// TIA Portal V19 export
FUNCTION "Analog_IN" : Void   // FC3, LAD
{ S7_Optimized_Access := 'TRUE' }
// stored: SetENOAutomatically false
BEGIN

REGION Network 1
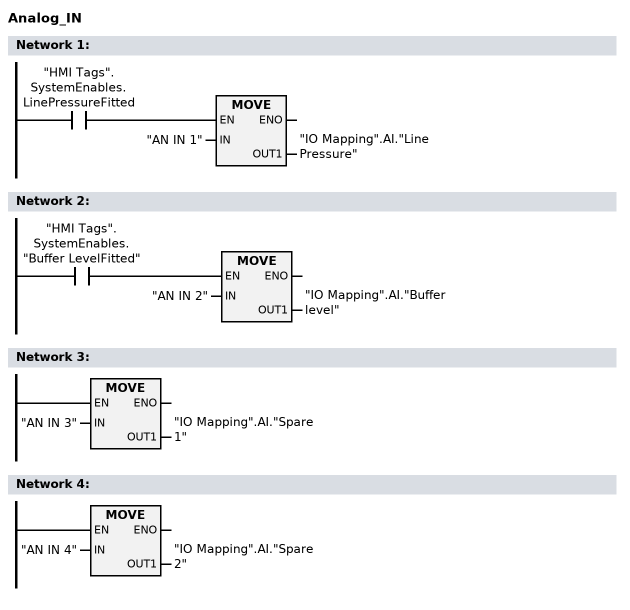
   RUNG wire#powerrail
      Contact( "HMI Tags".SystemEnables.LinePressureFitted )
      Move(in := "AN IN 1", out1 => "IO Mapping".AI."Line Pressure")
   END_RUNG
   // the same network as SCL:
   IF "HMI Tags".SystemEnables.LinePressureFitted THEN "IO Mapping".AI."Line Pressure" := "AN IN 1"; END_IF;
END_REGION

REGION Network 2
   RUNG wire#powerrail
      Contact( "HMI Tags".SystemEnables."Buffer LevelFitted" )
      Move(in := "AN IN 2", out1 => "IO Mapping".AI."Buffer level")
   END_RUNG
   // the same network as SCL:
   IF "HMI Tags".SystemEnables."Buffer LevelFitted" THEN "IO Mapping".AI."Buffer level" := "AN IN 2"; END_IF;
END_REGION

REGION Network 3
   RUNG wire#powerrail
      Move(in := "AN IN 3", out1 => "IO Mapping".AI."Spare 1")
   END_RUNG
   // the same network as SCL:
   "IO Mapping".AI."Spare 1" := "AN IN 3";
END_REGION

REGION Network 4
   RUNG wire#powerrail
      Move(in := "AN IN 4", out1 => "IO Mapping".AI."Spare 2")
   END_RUNG
   // the same network as SCL:
   "IO Mapping".AI."Spare 2" := "AN IN 4";
END_REGION
END_FUNCTION
